Staubli VAL3: Header.dtx

public num nMsgType
public num nCommType
public num nReplyCode
public num nData[12]
